// TIA Portal V20 export
DATA_BLOCK "Clock_DB"   // DB50
// stored: AutoNumber false, InstanceOfName Clock, InstanceOfType FB
"Clock"
   // VAR
   //    Var { ExternalAccessible := 'False'; ExternalVisible := 'False'; ExternalWritable := 'False'} : "TypeVar";
   //    opHoRun { ExternalAccessible := 'False'; ExternalVisible := 'False'; ExternalWritable := 'False'} : Bool;
   // END_VAR
BEGIN
END_DATA_BLOCK
